PROGRAM prgHouse
VAR PERSISTENT
	bEnableHouse		: BOOL;							//{#lynus.ag#()}
END_VAR
VAR
	fbHouse				: FB_HouseC_Power_Virtual;
	bHouseIsEnabled		: BOOL;							//{#lynus.ag#()}
	lrPowerHouse		: LREAL;						//{#lynus.ag#()}
END_VAR

fbHouse(
	bEnable:= bEnableHouse, 
	diNrOfEMS_IN:= prgEMS.fbEMS.diNrOfEMS_OUT, 
	bSetDefault:= , 
	lrCounterConsumptionSetDefault:= , 
	lrCounterProductionSetDefault:= , 
	stDataHouseC=> , 
	diNrOfHouseC_OUT=> );
	
lrPowerHouse := MAX(0,(prgPV.lrPowerPV + prgGrid.lrGridPower + prgBattery.lrPowerBattery - prgCS.lrPowerCS));
	bHouseIsEnabled := fbHouse.stDataHouseC.bEnabled;

END_PROGRAM

(* stored: Version 1.1.0.1, ProductVersion 3.1.4024.11
   POU prgHouse: Id {ff716a4d-a883-4467-b562-21fdcd65f5f8}, SpecialFunc None *)
